TEXTLIST SpindleStateList
  0 = 'SpindleIdle'
  1 = 'SpindleInitialization'
  2 = 'SpindleDisabled'
  3 = 'SpindleEnable'
  4 = 'SpindlePreMoving'
  5 = 'SpindleRotating'
  6 = 'SpindlePositioning'
  7 = 'SpindlePostMoving'
  8 = 'SpindleEmergency'
  9 = 'SpindleFault'
  10 = ''
   = ''
END_TEXTLIST

(* stored: Version 1.1.0.1, ProductVersion 3.1.4024.12
   TextList SpindleStateList: Id {c8ab4646-e2a6-48e9-a0da-383cda7a6729} *)
